RoboDK station: 03C - Option - Pick and Place.rdk

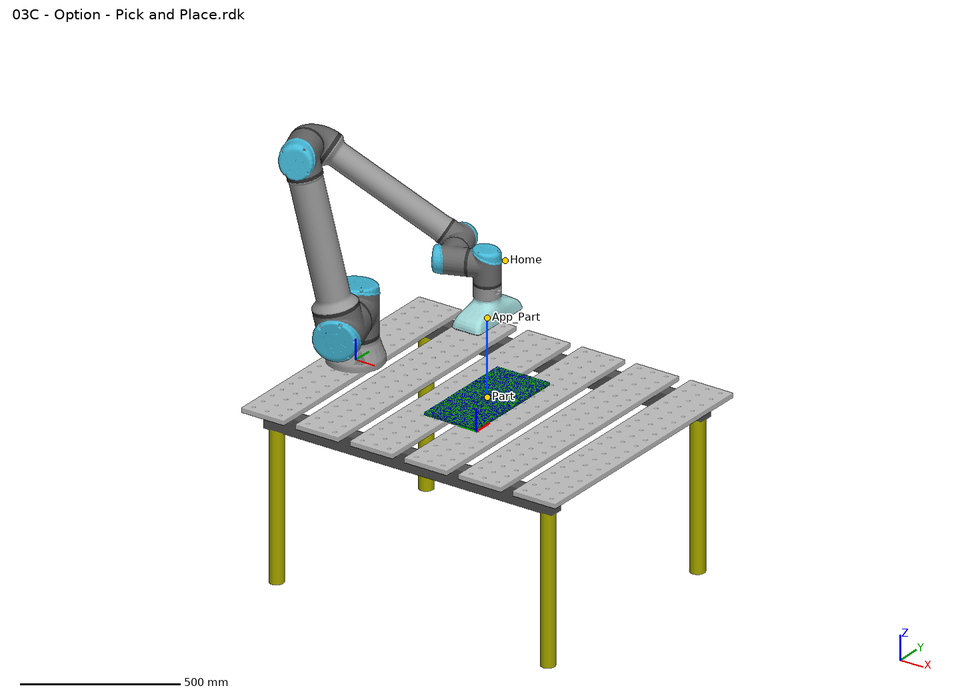
[picture v0: the station drawn from its stored meshes, robots at their saved joint values, targets as dots, program paths as lines]
Station 03C - Option - Pick and Place (saved by RoboDK 5.2.5). Poses are relative to the parent item; angles as X-Y-Z fixed-axis rotations.
Station parameters (name, value as stored): Palletizing Plugin
  - frame UR10e Base at (0, 0, 0) mm
    - robot UR10e: 6 axes, payload 10 kg, reach 1300 mm, repeatability 0.05 mm, weight 28.9 kg
        modified DH rows (alpha deg, a mm, theta deg, d mm): 0, 0, 0, 180.7; 90, 0, 180, 0; 0, 612.6, 0, 0; 0, 571.335, 0, 174.15; -90, 0, 0, 119.85; 90, 0, 180, 116.55
        joint limits [-360, -360, -360, -360, -360, -360] to [360, 360, 360, 360, 360, 360]; home [0, -90, -90, 0, 90, 0]; saved at [20.383, -77.494, -135.074, -57.433, 90, 20.383]
      - tool Vaccum, TCP at (0, 0, 69.67) mm, rotated rx 0 ry 0 rz 180 deg, size 247.5 x 110 x 75.9 mm, geometry from Vaccum.step
  - frame World at (0, 0, 0) mm
    - target Home (joint target) at (691.19, -174.15, 607.08) mm, rotated rx 180 ry 0 rz 90 deg; joints [0, -90, -90, -90, 90, 0] of UR10e
    - object Table at (500, 0, 0) mm, size 1193.8 x 965.2 x 609.6 mm, geometry from welding_table.sld
  - frame Part at (600, -200, 0) mm, rotated rx 0 ry 0 rz 90.06 deg
    - target Part (Cartesian target) at (200.11, 99.78, 10) mm, rotated rx 180 ry 0 rz -0.06 deg; joints [20.383, -110.98, -145.919, -13.101, 90, 20.383] of UR10e
    - target App_Part (Cartesian target) at (200.11, 99.78, 285) mm, rotated rx 180 ry 0 rz -0.06 deg; joints [20.383, -77.494, -135.074, -57.433, 90, 20.383] of UR10e
    - object PartBlue at (0, 0, 0) mm, size 400 x 200 x 10 mm, geometry from Part.step
    - object PartGreen at (0, 0, 0) mm, size 400 x 200 x 10 mm, geometry from Part.step
  - program PickPart (6 instructions, listed below)
  - program ReplaceObjects (1 instructions, listed below)
  - program GoHome (3 instructions, listed below)
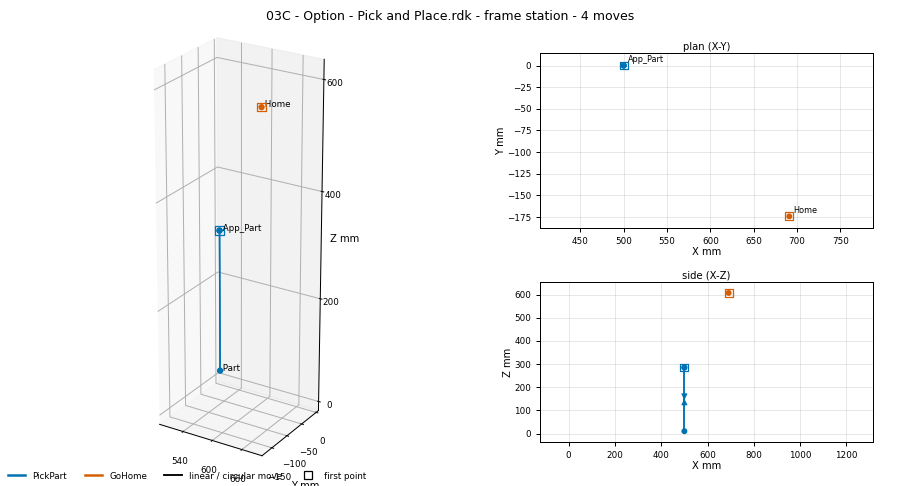
[picture p0: tool path of 03C - Option - Pick and Place.rdk in frame station, 4 of 4 moves have a stored position in this frame; points joined in program order, loops and branches not executed]

--- program PickPart (robot UR10e) ---
  Set Ref.: Part
  Set Tool: Vaccum
  MoveJ (App_Part)
  MoveL (Part)
  Attach to Vaccum
  MoveL (App_Part)

--- program ReplaceObjects (robot UR10e) ---
  Replace objects

--- program GoHome (robot UR10e) ---
  Set Ref.: World
  Set Tool: Vaccum
  MoveJ (Home)
